{attribute 'linkalways'} 
{attribute 'no_explicit_call' := 'This FB is a CLASS and must be accessed using methods or properties'}
{attribute 'enable_dynamic_creation'}
FUNCTION_BLOCK FINAL ADD_DWORD EXTENDS Node
VAR
	in1 : _DWORD(0);
	in2 : _DWORD(0);
	out : _DWORD(0);
END_VAR

METHOD PUBLIC Clone : I_Node
VAR
	pNode : POINTER TO ADD_DWORD;
END_VAR
pNode := __NEW(ADD_DWORD);
Clone := pNode^;
END_METHOD

METHOD FB_init : BOOL
VAR_INPUT
	bInitRetains : BOOL; // if TRUE, the retain variables are initialized (warm start / cold start)
	bInCopyCode : BOOL;  // if TRUE, the instance afterwards gets moved into the copy code (online change)
END_VAR
AddInput('in1',THIS^.in1);
AddInput('in2',THIS^.in2);
AddOutput('out', THIS^.out);
END_METHOD

METHOD PROTECTED OnExecute
VAR
END_VAR
out.Value := in1.Value + in2.Value;
END_METHOD

END_FUNCTION_BLOCK

(* stored: Version 1.1.0.1, ProductVersion 3.1.4024.15
   POU ADD_DWORD: Id {20eb1a2a-7597-4acb-92ab-f133f99f651d}, SpecialFunc None
   Folder Constructor: Id {679d6ff0-d1c7-4681-bb6a-e762dd9b28bc}
   Method Clone: Id {f2b01d31-7064-4e05-8322-760d57d42501}
   Method FB_init: Id {d5432840-4a97-4e48-b398-2dd7eaf0b426}
   Method OnExecute: Id {8ac264d9-5316-4da4-a0f6-e4edfb23c503} *)
